TYPE IoStd900 :
STRUCT	
	OutputPwm		AT %Q* : UINT;
	OutputPeriodPwm	AT %Q* : UINT;	
END_STRUCT
END_TYPE

(* stored: Version 1.1.0.1, ProductVersion 3.1.4024.4
   DUT IoStd900: Id {dec219e0-353b-48d1-945d-722f127d91e6} *)
